Omron CX-Programmer project NewProject (CX-Programmer 9.75)

# PLC NewPLC1: CQM1H CPU51

## Global symbols (name address type ; comment)
1.00 BOOL  ; Manual/Automatic
1.08 BOOL  ; MAN/Forward
1.09 BOOL  ; MAN/Revrese
1.12 BOOL  ; Man/Rotate Right
1.13 BOOL  ; Man/Rotate Left
1.14 BOOL  ; Man/Piston Up
1.15 BOOL  ; Man/Piston Down
LR4.01 BOOL  ; MEM/Forward
LR4.02 BOOL  ; MEM/Reverse
LR4.05 BOOL  ; MEM/Rotate Right
LR4.06 BOOL  ; MEM/Rotate Left
LR4.07 BOOL  ; MEM/Piston Up
LR4.08 BOOL  ; MEM/Piston Down

## Program NewProgram1 (no task)

### Section Section1

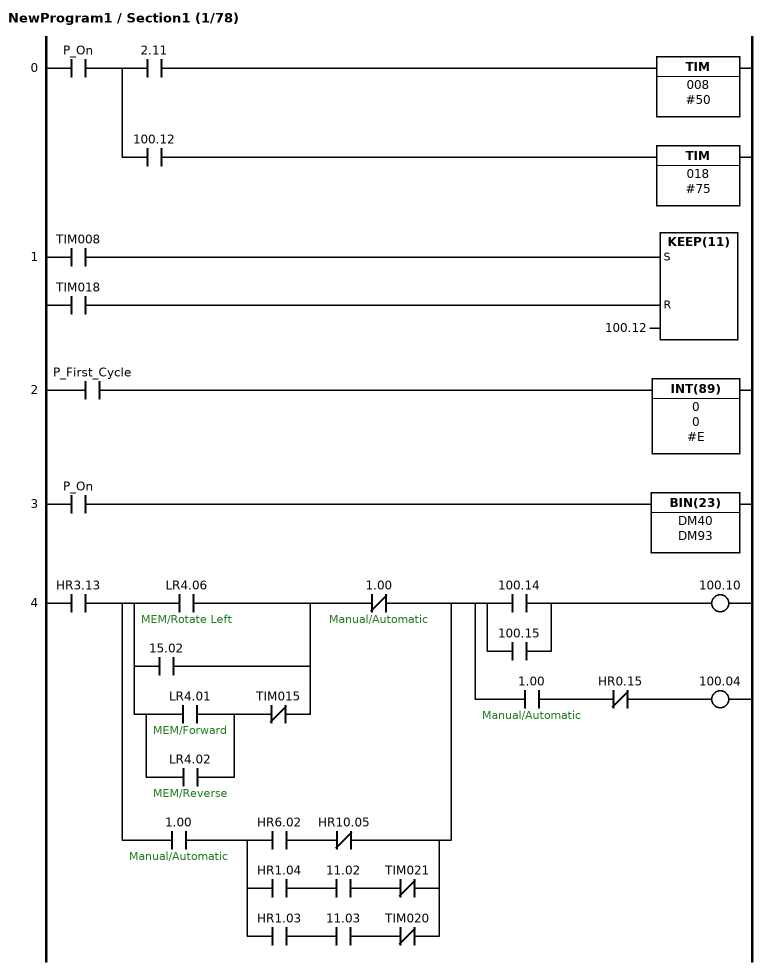
; rung 0
LD P_On
OUT TR0
AND 2.11
TIM 008 #50
LD TR0
AND 100.12
TIM 018 #75
; rung 1
LD TIM008
LD TIM018
KEEP(11) 100.12
; rung 2
LD P_First_Cycle
INT(89) 0 0 #E
; rung 3
LD P_On
BIN(23) DM40 DM93
; rung 4
LD HR3.13
LD LR4.06  ; MEM/Rotate Left
OR 15.02
LD LR4.01  ; MEM/Forward
OR LR4.02  ; MEM/Reverse
ANDNOT TIM015
ORLD
ANDNOT 1.00  ; Manual/Automatic
LD 1.00  ; Manual/Automatic
LD HR6.02
ANDNOT HR10.05
LD HR1.04
AND 11.02
ANDNOT TIM021
ORLD
LD HR1.03
AND 11.03
ANDNOT TIM020
ORLD
ANDLD
ORLD
ANDLD
OUT TR0
LD 100.14
OR 100.15
ANDLD
OUT 100.10
LD TR0
AND 1.00  ; Manual/Automatic
ANDNOT HR0.15
OUT 100.04

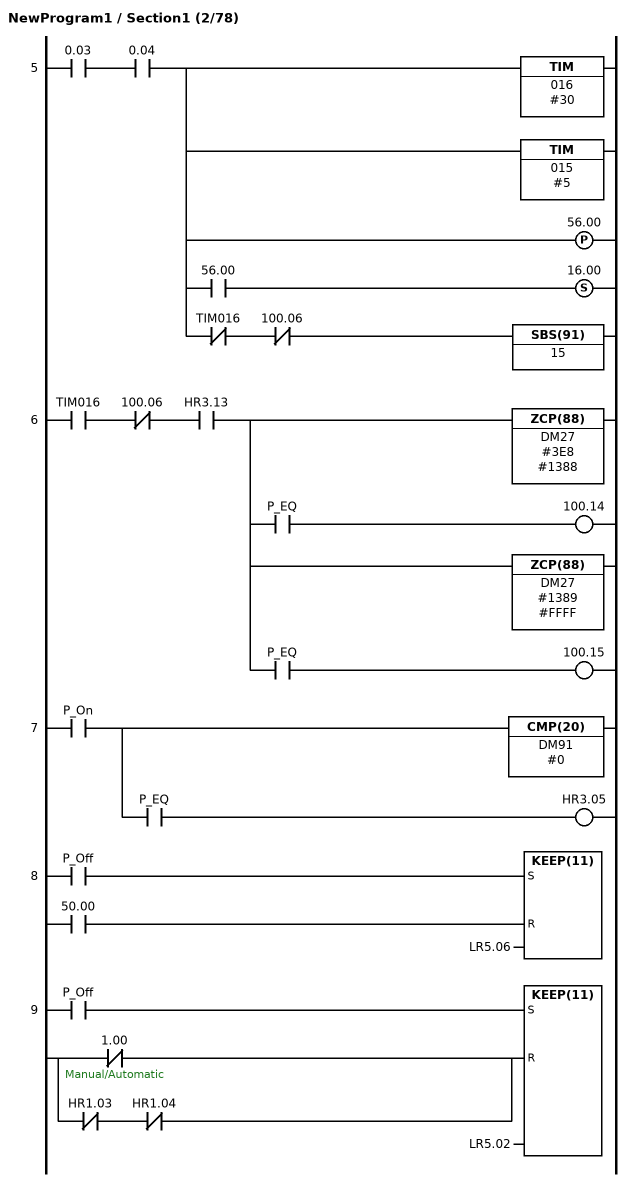
; rung 5
LD 0.03
AND 0.04
OUT TR0
TIM 016 #30
TIM 015 #5
DIFU(13) 56.00
AND 56.00
SET 16.00
LD TR0
ANDNOT TIM016
ANDNOT 100.06
SBS(91) 15
; rung 6
LD TIM016
ANDNOT 100.06
AND HR3.13
OUT TR0
ZCP(88) DM27 #3E8 #1388
AND P_EQ
OUT 100.14
LD TR0
ZCP(88) DM27 #1389 #FFFF
AND P_EQ
OUT 100.15
; rung 7
LD P_On
CMP(20) DM91 #0
AND P_EQ
OUT HR3.05
; rung 8
LD P_Off
LD 50.00
KEEP(11) LR5.06
; rung 9
LD P_Off
LDNOT 1.00  ; Manual/Automatic
LDNOT HR1.03
ANDNOT HR1.04
ORLD
KEEP(11) LR5.02

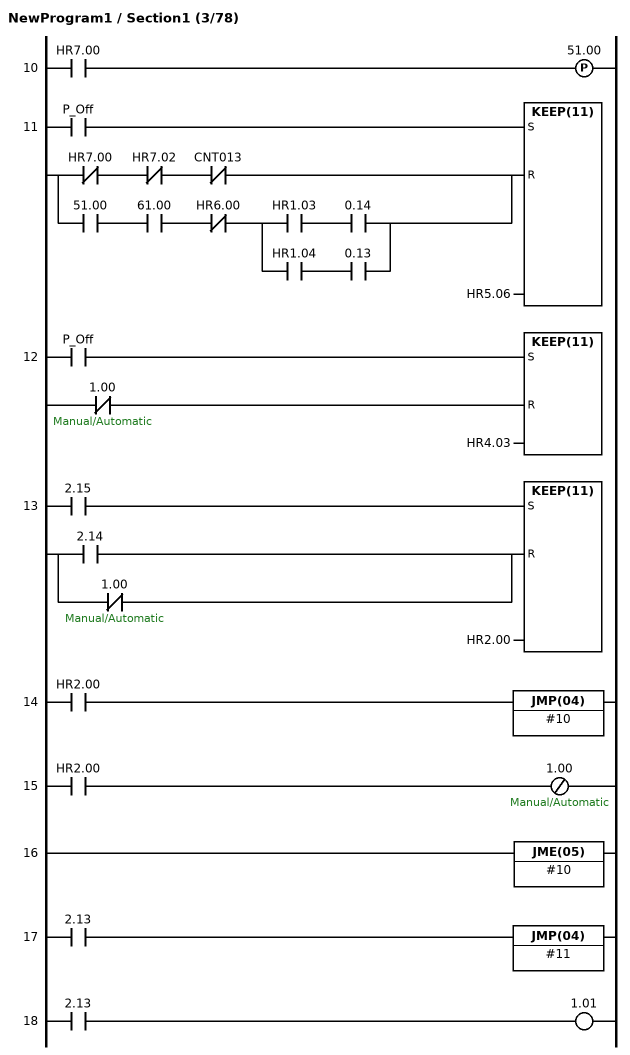
; rung 10
LD HR7.00
DIFU(13) 51.00
; rung 11
LD P_Off
LDNOT HR7.00
ANDNOT HR7.02
ANDNOT CNT013
LD 51.00
AND 61.00
ANDNOT HR6.00
LD HR1.03
AND 0.14
LD HR1.04
AND 0.13
ORLD
ANDLD
ORLD
KEEP(11) HR5.06
; rung 12
LD P_Off
LDNOT 1.00  ; Manual/Automatic
KEEP(11) HR4.03
; rung 13
LD 2.15
LD 2.14
ORNOT 1.00  ; Manual/Automatic
KEEP(11) HR2.00
; rung 14
LD HR2.00
JMP(04) #10
; rung 15
LD HR2.00
OUTNOT 1.00  ; Manual/Automatic
; rung 16
JME(05) #10
; rung 17
LD 2.13
JMP(04) #11
; rung 18
LD 2.13
OUT 1.01

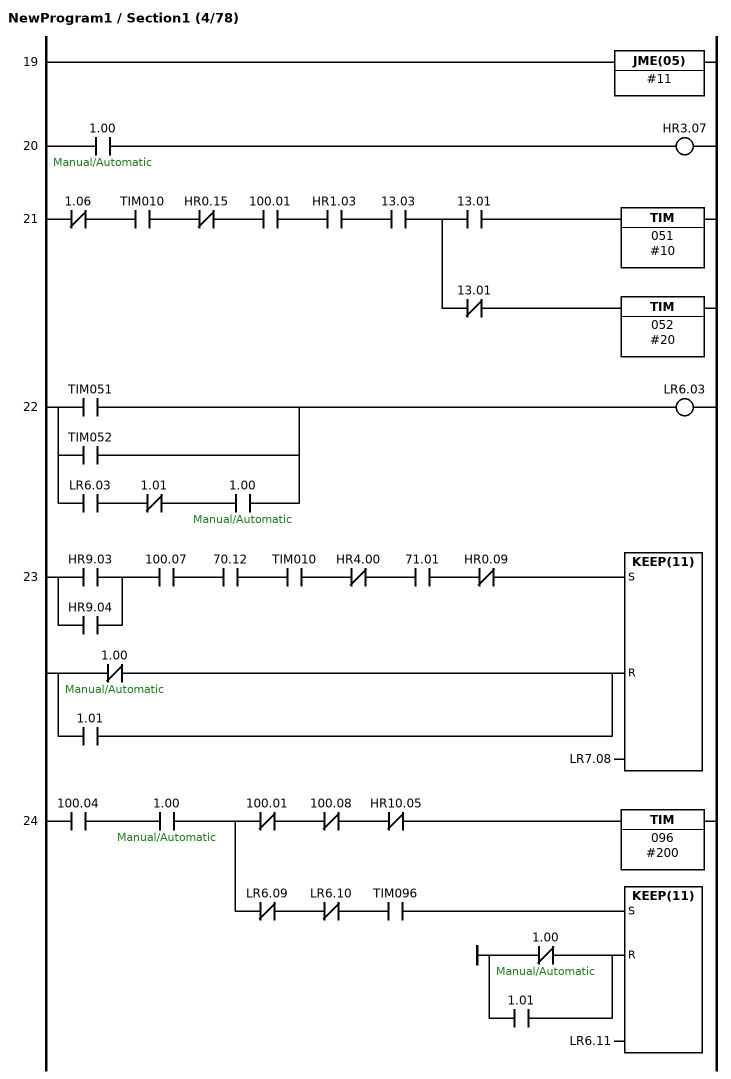
; rung 19
JME(05) #11
; rung 20
LD 1.00  ; Manual/Automatic
OUT HR3.07
; rung 21
LDNOT 1.06
AND TIM010
ANDNOT HR0.15
AND 100.01
AND HR1.03
AND 13.03
OUT TR0
AND 13.01
TIM 051 #10
LD TR0
ANDNOT 13.01
TIM 052 #20
; rung 22
LD TIM051
OR TIM052
LD LR6.03
ANDNOT 1.01
AND 1.00  ; Manual/Automatic
ORLD
OUT LR6.03
; rung 23
LD HR9.03
OR HR9.04
AND 100.07
AND 70.12
AND TIM010
ANDNOT HR4.00
AND 71.01
ANDNOT HR0.09
LDNOT 1.00  ; Manual/Automatic
OR 1.01
KEEP(11) LR7.08
; rung 24
LD 100.04
AND 1.00  ; Manual/Automatic
OUT TR0
ANDNOT 100.01
ANDNOT 100.08
ANDNOT HR10.05
TIM 096 #200
LD TR0
ANDNOT LR6.09
ANDNOT LR6.10
AND TIM096
LDNOT 1.00  ; Manual/Automatic
OR 1.01
KEEP(11) LR6.11

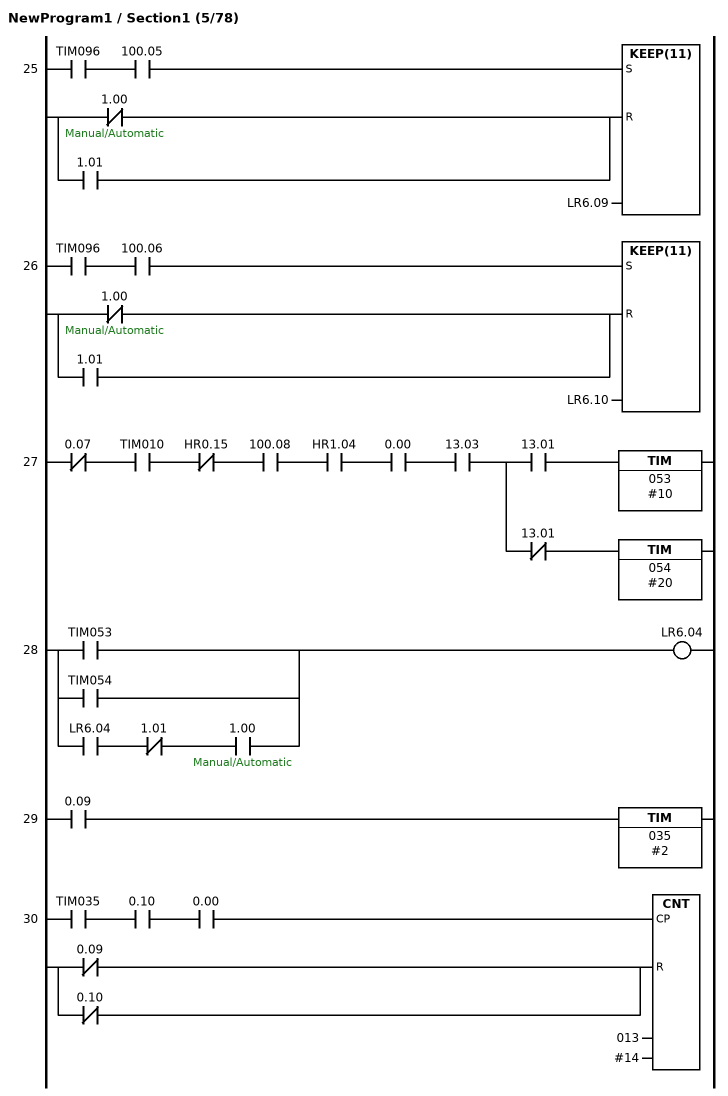
; rung 25
LD TIM096
AND 100.05
LDNOT 1.00  ; Manual/Automatic
OR 1.01
KEEP(11) LR6.09
; rung 26
LD TIM096
AND 100.06
LDNOT 1.00  ; Manual/Automatic
OR 1.01
KEEP(11) LR6.10
; rung 27
LDNOT 0.07
AND TIM010
ANDNOT HR0.15
AND 100.08
AND HR1.04
AND 0.00
AND 13.03
OUT TR0
AND 13.01
TIM 053 #10
LD TR0
ANDNOT 13.01
TIM 054 #20
; rung 28
LD TIM053
OR TIM054
LD LR6.04
ANDNOT 1.01
AND 1.00  ; Manual/Automatic
ORLD
OUT LR6.04
; rung 29
LD 0.09
TIM 035 #2
; rung 30
LD TIM035
AND 0.10
AND 0.00
LDNOT 0.09
ORNOT 0.10
CNT 013 #14

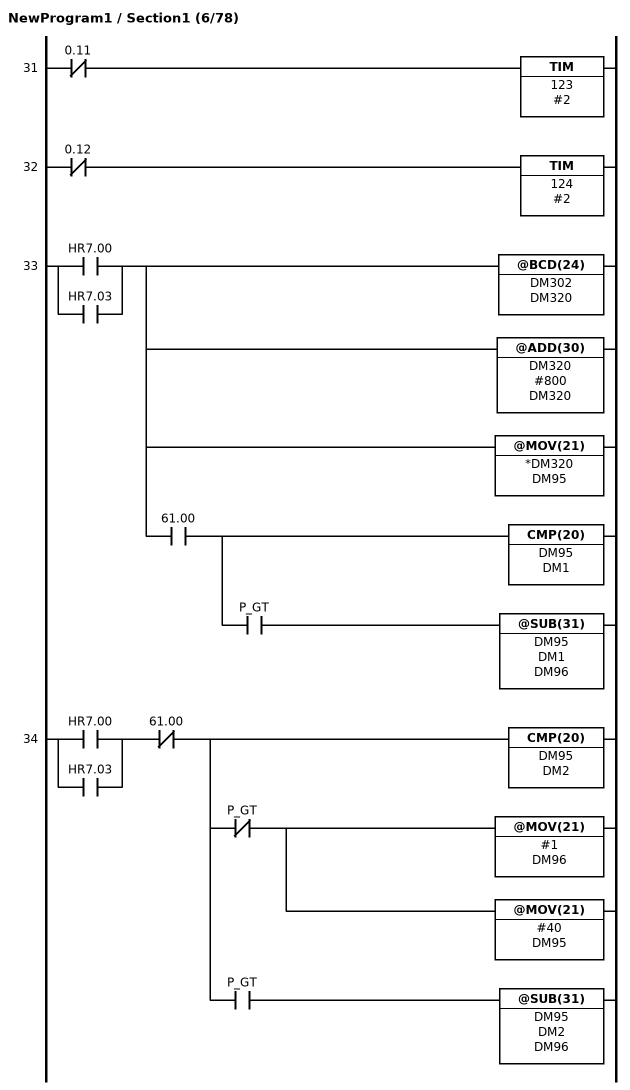
; rung 31
LDNOT 0.11
TIM 123 #2
; rung 32
LDNOT 0.12
TIM 124 #2
; rung 33
LD HR7.00
OR HR7.03
@BCD(24) DM302 DM320
@ADD(30) DM320 #800 DM320
@MOV(21) *DM320 DM95
AND 61.00
CMP(20) DM95 DM1
AND P_GT
@SUB(31) DM95 DM1 DM96
; rung 34
LD HR7.00
OR HR7.03
ANDNOT 61.00
OUT TR0
CMP(20) DM95 DM2
ANDNOT P_GT
@MOV(21) #1 DM96
@MOV(21) #40 DM95
LD TR0
AND P_GT
@SUB(31) DM95 DM2 DM96

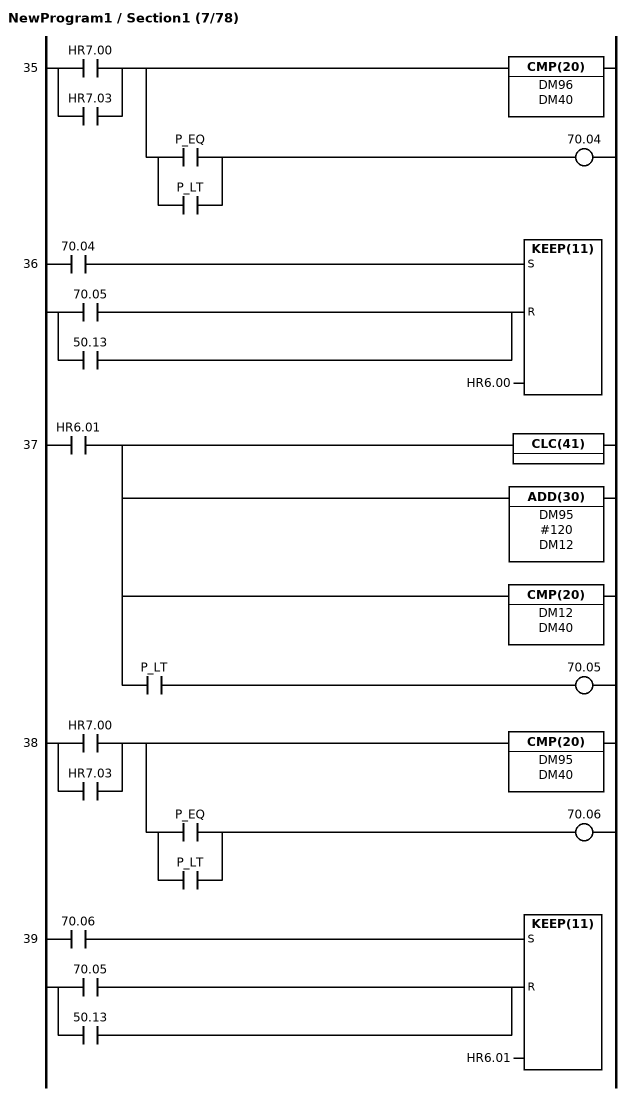
; rung 35
LD HR7.00
OR HR7.03
CMP(20) DM96 DM40
LD P_EQ
OR P_LT
ANDLD
OUT 70.04
; rung 36
LD 70.04
LD 70.05
OR 50.13
KEEP(11) HR6.00
; rung 37
LD HR6.01
CLC(41)
ADD(30) DM95 #120 DM12
CMP(20) DM12 DM40
AND P_LT
OUT 70.05
; rung 38
LD HR7.00
OR HR7.03
CMP(20) DM95 DM40
LD P_EQ
OR P_LT
ANDLD
OUT 70.06
; rung 39
LD 70.06
LD 70.05
OR 50.13
KEEP(11) HR6.01

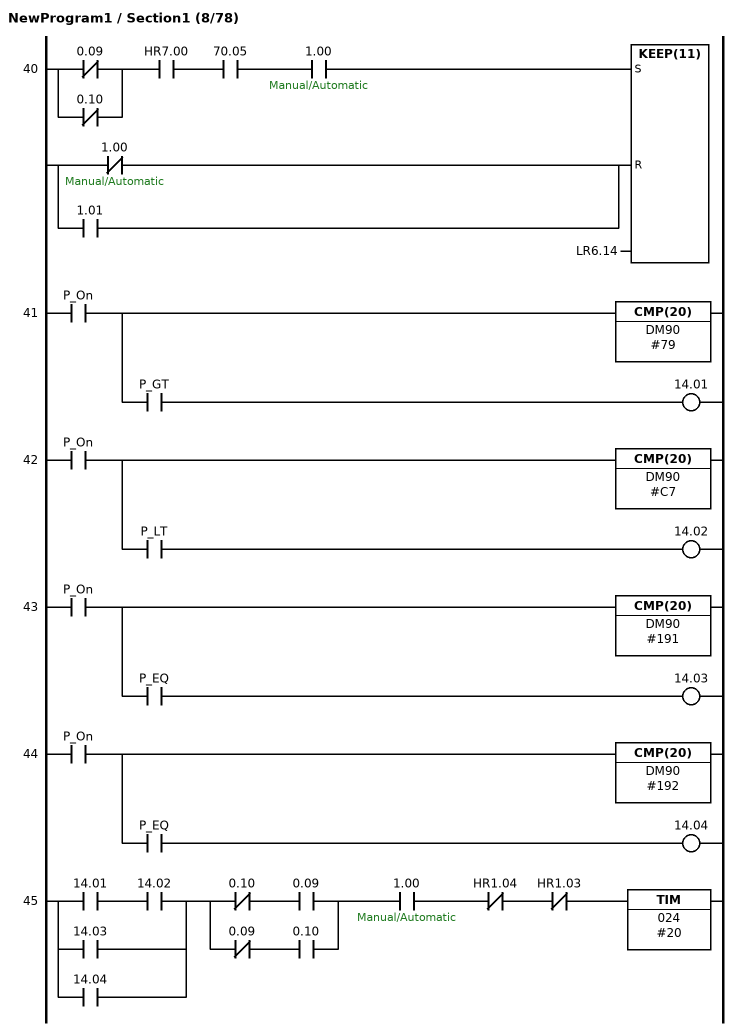
; rung 40
LDNOT 0.09
ORNOT 0.10
AND HR7.00
AND 70.05
AND 1.00  ; Manual/Automatic
LDNOT 1.00  ; Manual/Automatic
OR 1.01
KEEP(11) LR6.14
; rung 41
LD P_On
CMP(20) DM90 #79
AND P_GT
OUT 14.01
; rung 42
LD P_On
CMP(20) DM90 #C7
AND P_LT
OUT 14.02
; rung 43
LD P_On
CMP(20) DM90 #191
AND P_EQ
OUT 14.03
; rung 44
LD P_On
CMP(20) DM90 #192
AND P_EQ
OUT 14.04
; rung 45
LD 14.01
AND 14.02
OR 14.03
OR 14.04
LDNOT 0.10
AND 0.09
LDNOT 0.09
AND 0.10
ORLD
ANDLD
AND 1.00  ; Manual/Automatic
ANDNOT HR1.04
ANDNOT HR1.03
TIM 024 #20

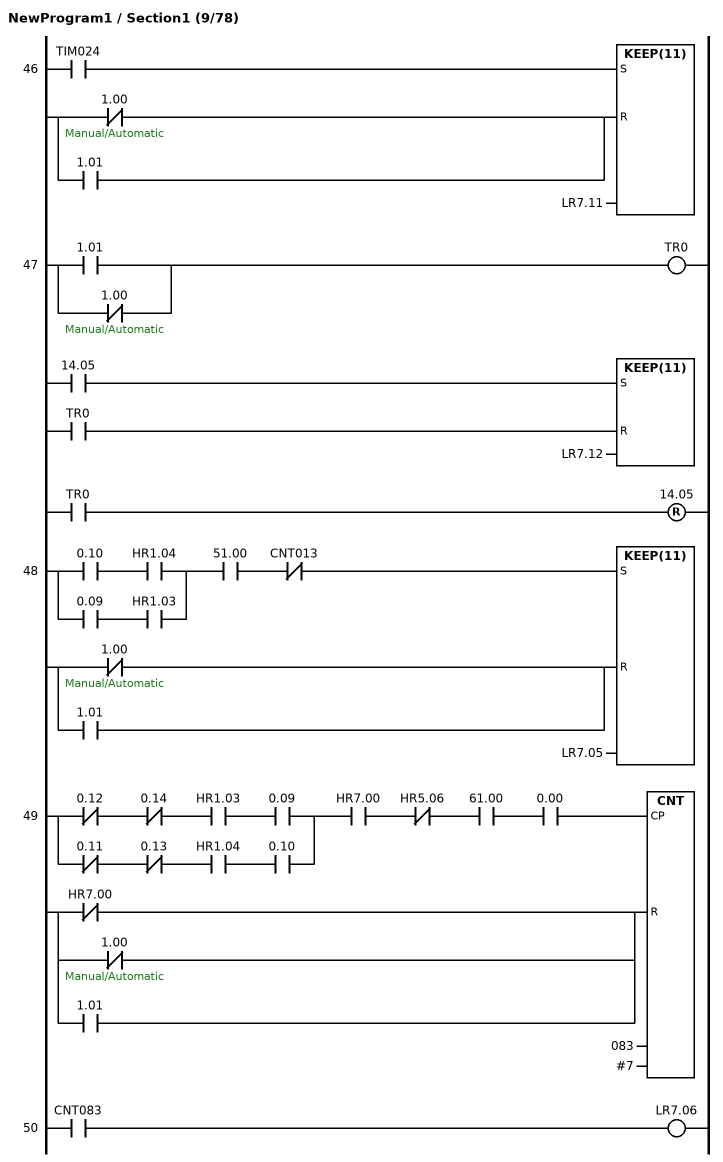
; rung 46
LD TIM024
LDNOT 1.00  ; Manual/Automatic
OR 1.01
KEEP(11) LR7.11
; rung 47
LD 14.05
LD 1.01
ORNOT 1.00  ; Manual/Automatic
OUT TR0
KEEP(11) LR7.12
LD TR0
RSET 14.05
; rung 48
LD 0.10
AND HR1.04
LD 0.09
AND HR1.03
ORLD
AND 51.00
ANDNOT CNT013
LDNOT 1.00  ; Manual/Automatic
OR 1.01
KEEP(11) LR7.05
; rung 49
LDNOT 0.12
ANDNOT 0.14
AND HR1.03
AND 0.09
LDNOT 0.11
ANDNOT 0.13
AND HR1.04
AND 0.10
ORLD
AND HR7.00
ANDNOT HR5.06
AND 61.00
AND 0.00
LDNOT HR7.00
ORNOT 1.00  ; Manual/Automatic
OR 1.01
CNT 083 #7
; rung 50
LD CNT083
OUT LR7.06

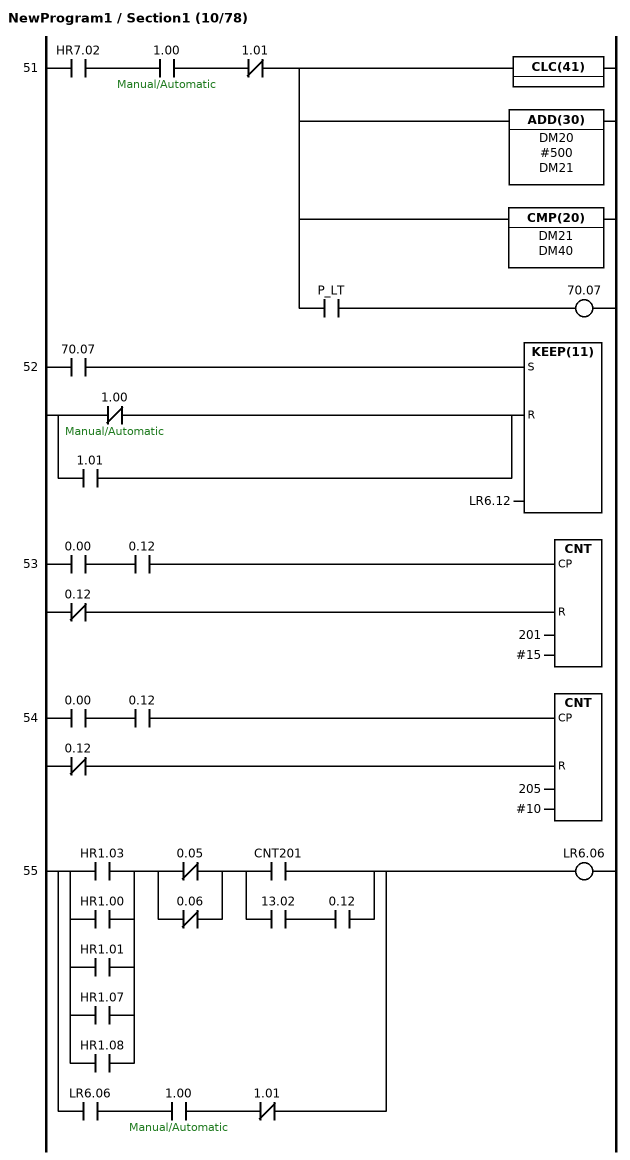
; rung 51
LD HR7.02
AND 1.00  ; Manual/Automatic
ANDNOT 1.01
CLC(41)
ADD(30) DM20 #500 DM21
CMP(20) DM21 DM40
AND P_LT
OUT 70.07
; rung 52
LD 70.07
LDNOT 1.00  ; Manual/Automatic
OR 1.01
KEEP(11) LR6.12
; rung 53
LD 0.00
AND 0.12
LDNOT 0.12
CNT 201 #15
; rung 54
LD 0.00
AND 0.12
LDNOT 0.12
CNT 205 #10
; rung 55
LD HR1.03
OR HR1.00
OR HR1.01
OR HR1.07
OR HR1.08
LDNOT 0.05
ORNOT 0.06
ANDLD
LD CNT201
LD 13.02
AND 0.12
ORLD
ANDLD
LD LR6.06
AND 1.00  ; Manual/Automatic
ANDNOT 1.01
ORLD
OUT LR6.06

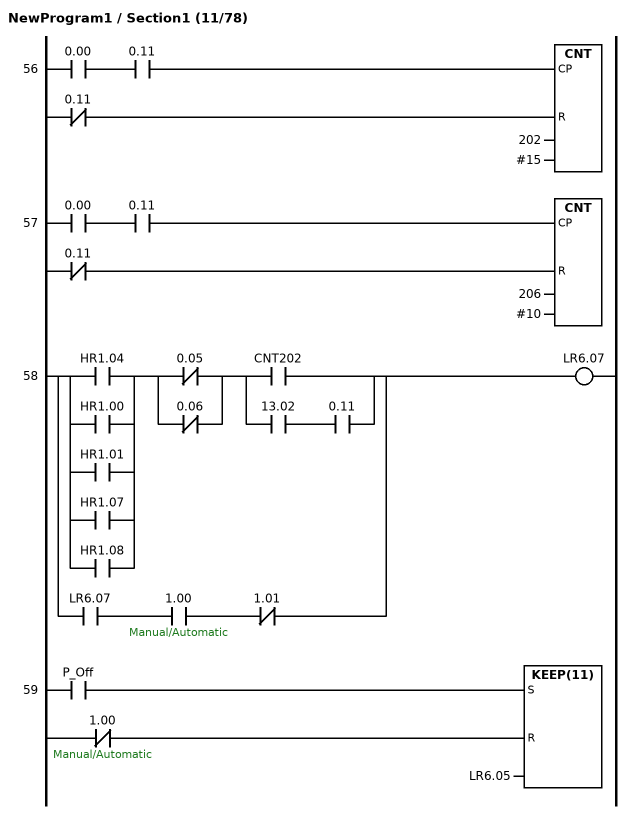
; rung 56
LD 0.00
AND 0.11
LDNOT 0.11
CNT 202 #15
; rung 57
LD 0.00
AND 0.11
LDNOT 0.11
CNT 206 #10
; rung 58
LD HR1.04
OR HR1.00
OR HR1.01
OR HR1.07
OR HR1.08
LDNOT 0.05
ORNOT 0.06
ANDLD
LD CNT202
LD 13.02
AND 0.11
ORLD
ANDLD
LD LR6.07
AND 1.00  ; Manual/Automatic
ANDNOT 1.01
ORLD
OUT LR6.07
; rung 59
LD P_Off
LDNOT 1.00  ; Manual/Automatic
KEEP(11) LR6.05

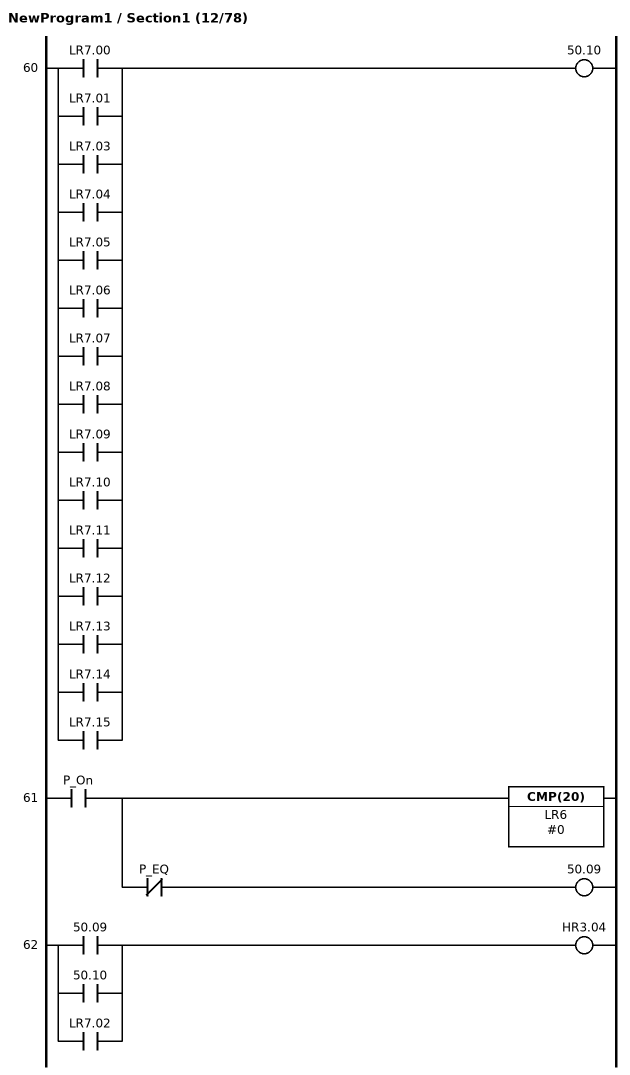
; rung 60
LD LR7.00
OR LR7.01
OR LR7.03
OR LR7.04
OR LR7.05
OR LR7.06
OR LR7.07
OR LR7.08
OR LR7.09
OR LR7.10
OR LR7.11
OR LR7.12
OR LR7.13
OR LR7.14
OR LR7.15
OUT 50.10
; rung 61
LD P_On
CMP(20) LR6 #0
ANDNOT P_EQ
OUT 50.09
; rung 62
LD 50.09
OR 50.10
OR LR7.02
OUT HR3.04

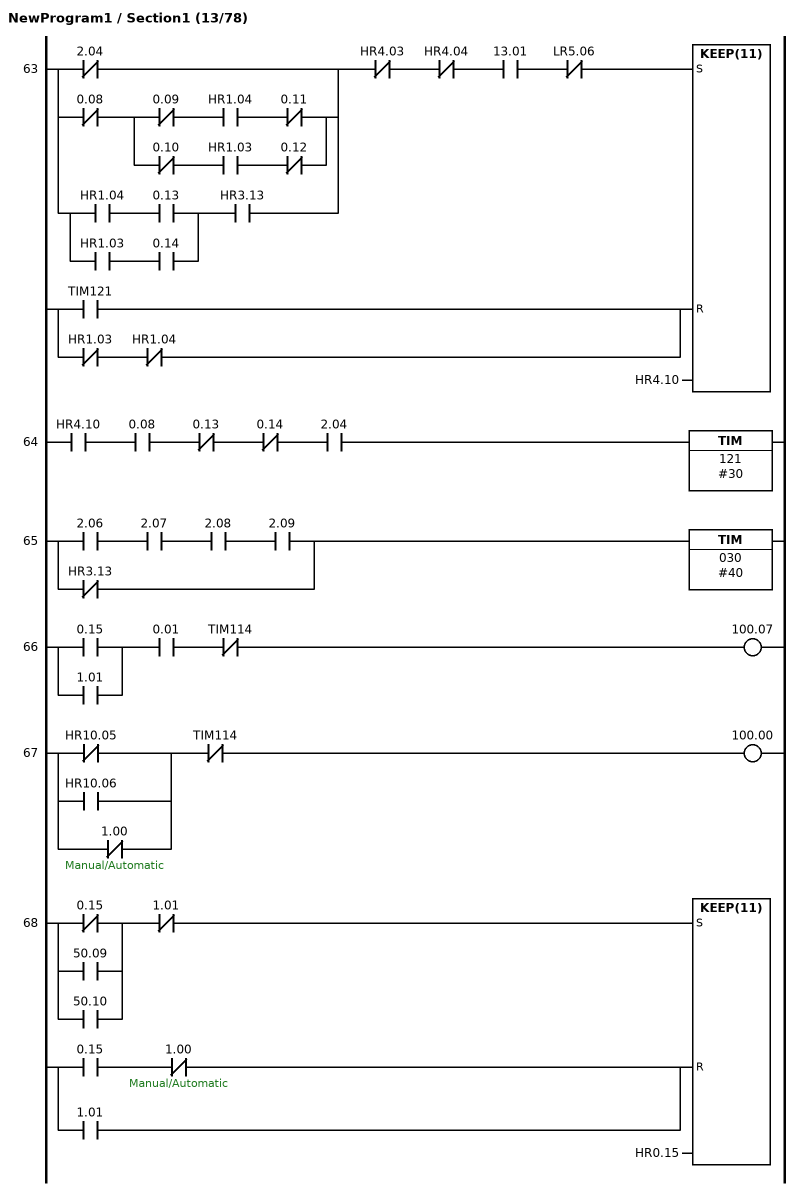
; rung 63
LDNOT 2.04
LDNOT 0.08
LDNOT 0.09
AND HR1.04
ANDNOT 0.11
LDNOT 0.10
AND HR1.03
ANDNOT 0.12
ORLD
ANDLD
ORLD
LD HR1.04
AND 0.13
LD HR1.03
AND 0.14
ORLD
AND HR3.13
ORLD
ANDNOT HR4.03
ANDNOT HR4.04
AND 13.01
ANDNOT LR5.06
LD TIM121
LDNOT HR1.03
ANDNOT HR1.04
ORLD
KEEP(11) HR4.10
; rung 64
LD HR4.10
AND 0.08
ANDNOT 0.13
ANDNOT 0.14
AND 2.04
TIM 121 #30
; rung 65
LD 2.06
AND 2.07
AND 2.08
AND 2.09
ORNOT HR3.13
TIM 030 #40
; rung 66
LD 0.15
OR 1.01
AND 0.01
ANDNOT TIM114
OUT 100.07
; rung 67
LDNOT HR10.05
OR HR10.06
ORNOT 1.00  ; Manual/Automatic
ANDNOT TIM114
OUT 100.00
; rung 68
LDNOT 0.15
OR 50.09
OR 50.10
ANDNOT 1.01
LD 0.15
ANDNOT 1.00  ; Manual/Automatic
OR 1.01
KEEP(11) HR0.15

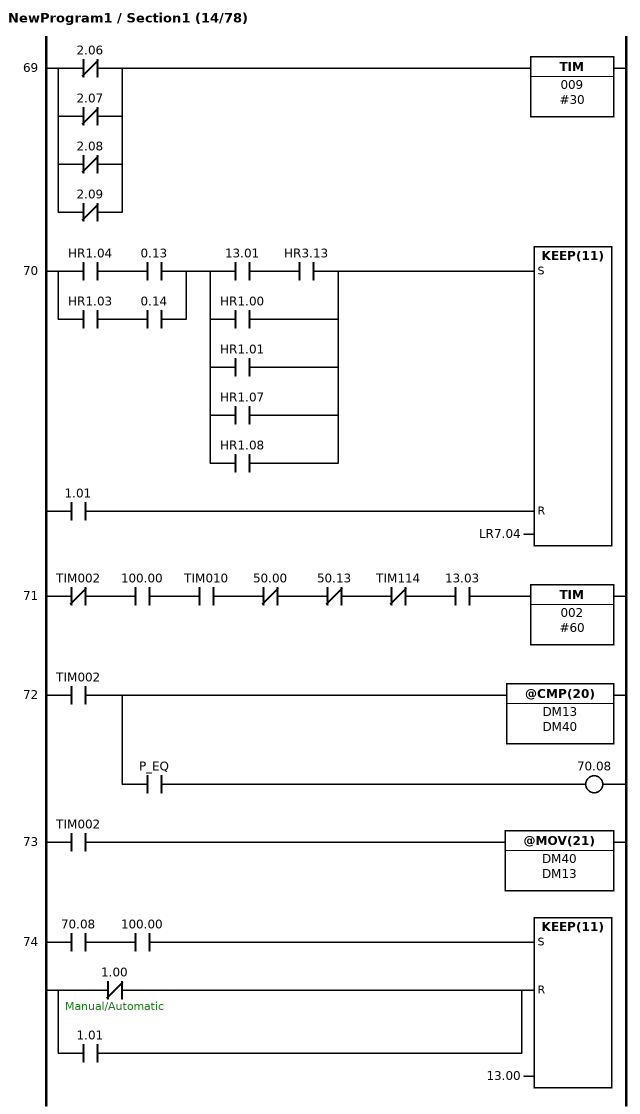
; rung 69
LDNOT 2.06
ORNOT 2.07
ORNOT 2.08
ORNOT 2.09
TIM 009 #30
; rung 70
LD HR1.04
AND 0.13
LD HR1.03
AND 0.14
ORLD
LD 13.01
AND HR3.13
OR HR1.00
OR HR1.01
OR HR1.07
OR HR1.08
ANDLD
LD 1.01
KEEP(11) LR7.04
; rung 71
LDNOT TIM002
AND 100.00
AND TIM010
ANDNOT 50.00
ANDNOT 50.13
ANDNOT TIM114
AND 13.03
TIM 002 #60
; rung 72
LD TIM002
@CMP(20) DM13 DM40
AND P_EQ
OUT 70.08
; rung 73
LD TIM002
@MOV(21) DM40 DM13
; rung 74
LD 70.08
AND 100.00
LDNOT 1.00  ; Manual/Automatic
OR 1.01
KEEP(11) 13.00

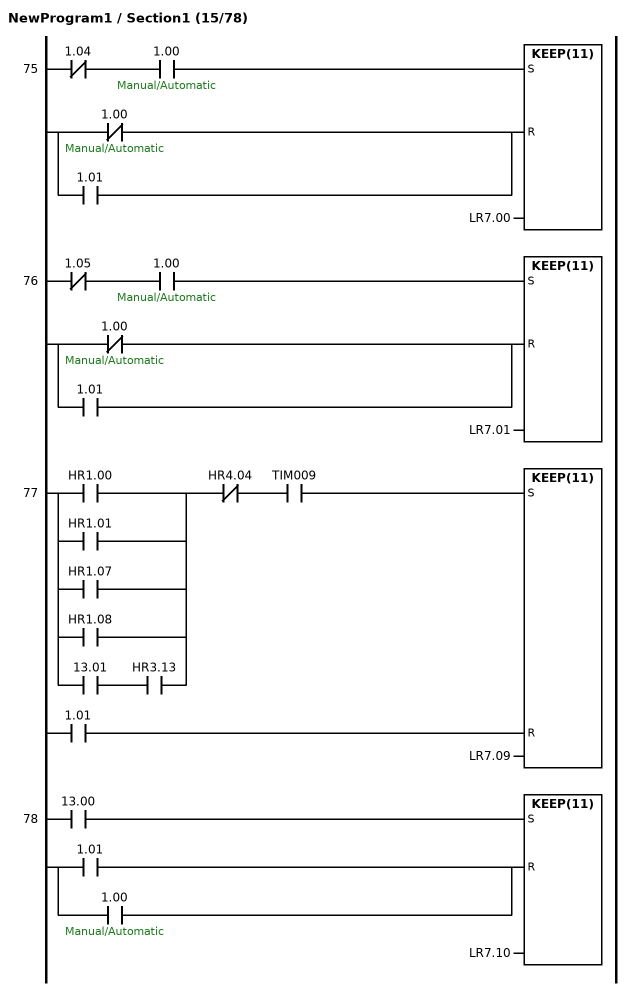
; rung 75
LDNOT 1.04
AND 1.00  ; Manual/Automatic
LDNOT 1.00  ; Manual/Automatic
OR 1.01
KEEP(11) LR7.00
; rung 76
LDNOT 1.05
AND 1.00  ; Manual/Automatic
LDNOT 1.00  ; Manual/Automatic
OR 1.01
KEEP(11) LR7.01
; rung 77
LD HR1.00
OR HR1.01
OR HR1.07
OR HR1.08
LD 13.01
AND HR3.13
ORLD
ANDNOT HR4.04
AND TIM009
LD 1.01
KEEP(11) LR7.09
; rung 78
LD 13.00
LD 1.01
OR 1.00  ; Manual/Automatic
KEEP(11) LR7.10

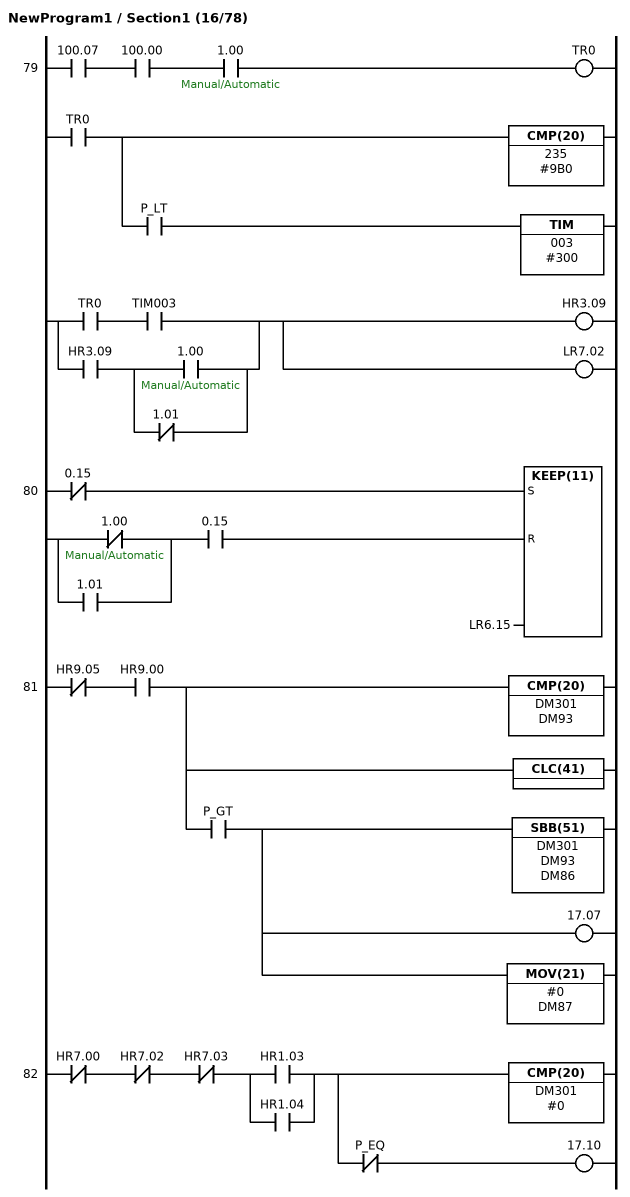
; rung 79
LD 100.07
AND 100.00
AND 1.00  ; Manual/Automatic
OUT TR0
CMP(20) 235 #9B0
AND P_LT
TIM 003 #300
LD TR0
AND TIM003
LD HR3.09
LD 1.00  ; Manual/Automatic
ORNOT 1.01
ANDLD
ORLD
OUT HR3.09
OUT LR7.02
; rung 80
LDNOT 0.15
LDNOT 1.00  ; Manual/Automatic
OR 1.01
AND 0.15
KEEP(11) LR6.15
; rung 81
LDNOT HR9.05
AND HR9.00
CMP(20) DM301 DM93
CLC(41)
AND P_GT
SBB(51) DM301 DM93 DM86
OUT 17.07
MOV(21) #0 DM87
; rung 82
LDNOT HR7.00
ANDNOT HR7.02
ANDNOT HR7.03
LD HR1.03
OR HR1.04
ANDLD
CMP(20) DM301 #0
ANDNOT P_EQ
OUT 17.10

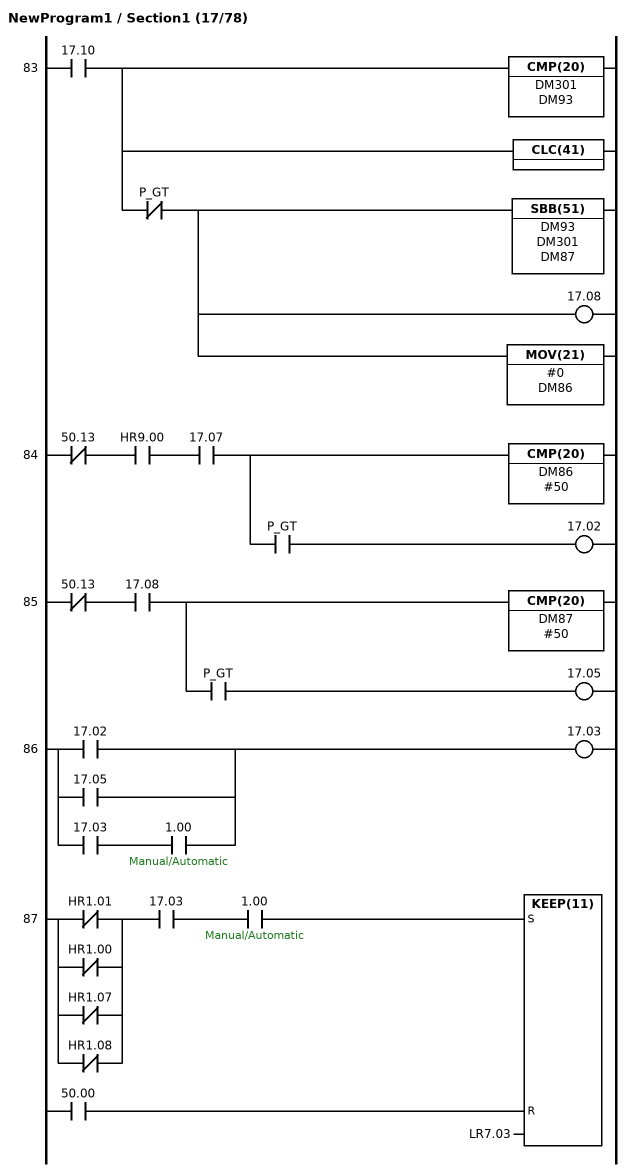
; rung 83
LD 17.10
CMP(20) DM301 DM93
CLC(41)
ANDNOT P_GT
SBB(51) DM93 DM301 DM87
OUT 17.08
MOV(21) #0 DM86
; rung 84
LDNOT 50.13
AND HR9.00
AND 17.07
CMP(20) DM86 #50
AND P_GT
OUT 17.02
; rung 85
LDNOT 50.13
AND 17.08
CMP(20) DM87 #50
AND P_GT
OUT 17.05
; rung 86
LD 17.02
OR 17.05
LD 17.03
AND 1.00  ; Manual/Automatic
ORLD
OUT 17.03
; rung 87
LDNOT HR1.01
ORNOT HR1.00
ORNOT HR1.07
ORNOT HR1.08
AND 17.03
AND 1.00  ; Manual/Automatic
LD 50.00
KEEP(11) LR7.03

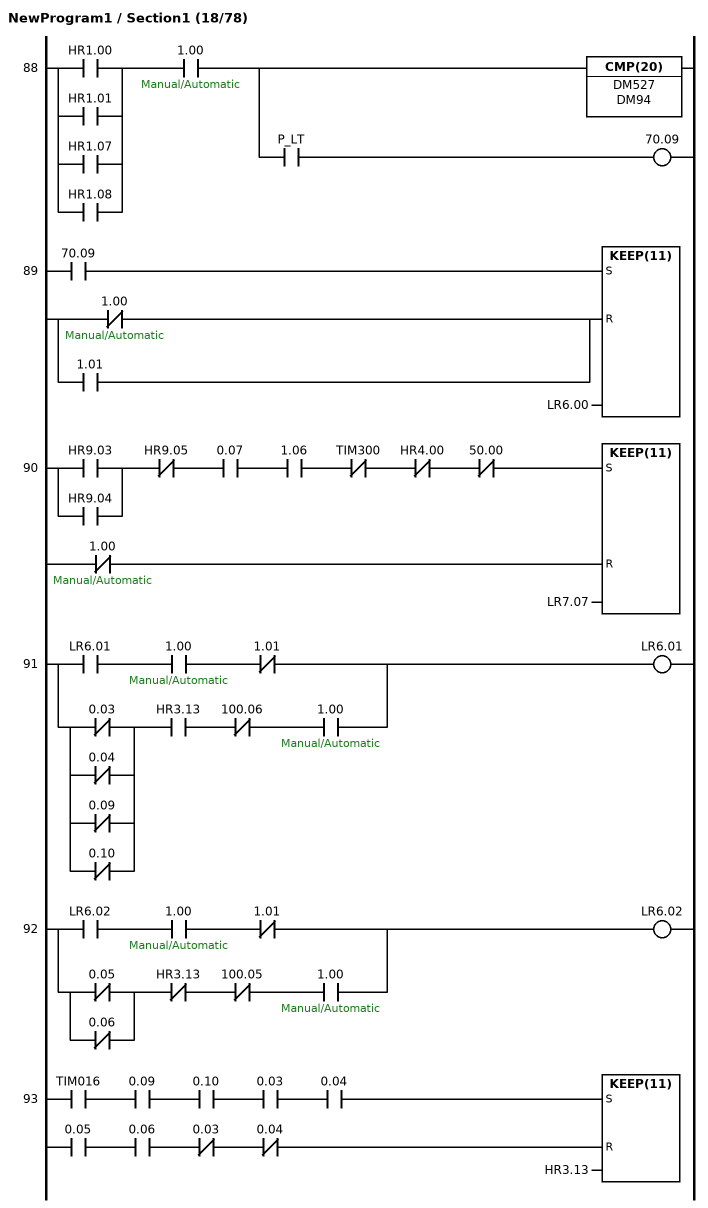
; rung 88
LD HR1.00
OR HR1.01
OR HR1.07
OR HR1.08
AND 1.00  ; Manual/Automatic
CMP(20) DM527 DM94
AND P_LT
OUT 70.09
; rung 89
LD 70.09
LDNOT 1.00  ; Manual/Automatic
OR 1.01
KEEP(11) LR6.00
; rung 90
LD HR9.03
OR HR9.04
ANDNOT HR9.05
AND 0.07
AND 1.06
ANDNOT TIM300
ANDNOT HR4.00
ANDNOT 50.00
LDNOT 1.00  ; Manual/Automatic
KEEP(11) LR7.07
; rung 91
LD LR6.01
AND 1.00  ; Manual/Automatic
ANDNOT 1.01
LDNOT 0.03
ORNOT 0.04
ORNOT 0.09
ORNOT 0.10
AND HR3.13
ANDNOT 100.06
AND 1.00  ; Manual/Automatic
ORLD
OUT LR6.01
; rung 92
LD LR6.02
AND 1.00  ; Manual/Automatic
ANDNOT 1.01
LDNOT 0.05
ORNOT 0.06
ANDNOT HR3.13
ANDNOT 100.05
AND 1.00  ; Manual/Automatic
ORLD
OUT LR6.02
; rung 93
LD TIM016
AND 0.09
AND 0.10
AND 0.03
AND 0.04
LD 0.05
AND 0.06
ANDNOT 0.03
ANDNOT 0.04
KEEP(11) HR3.13

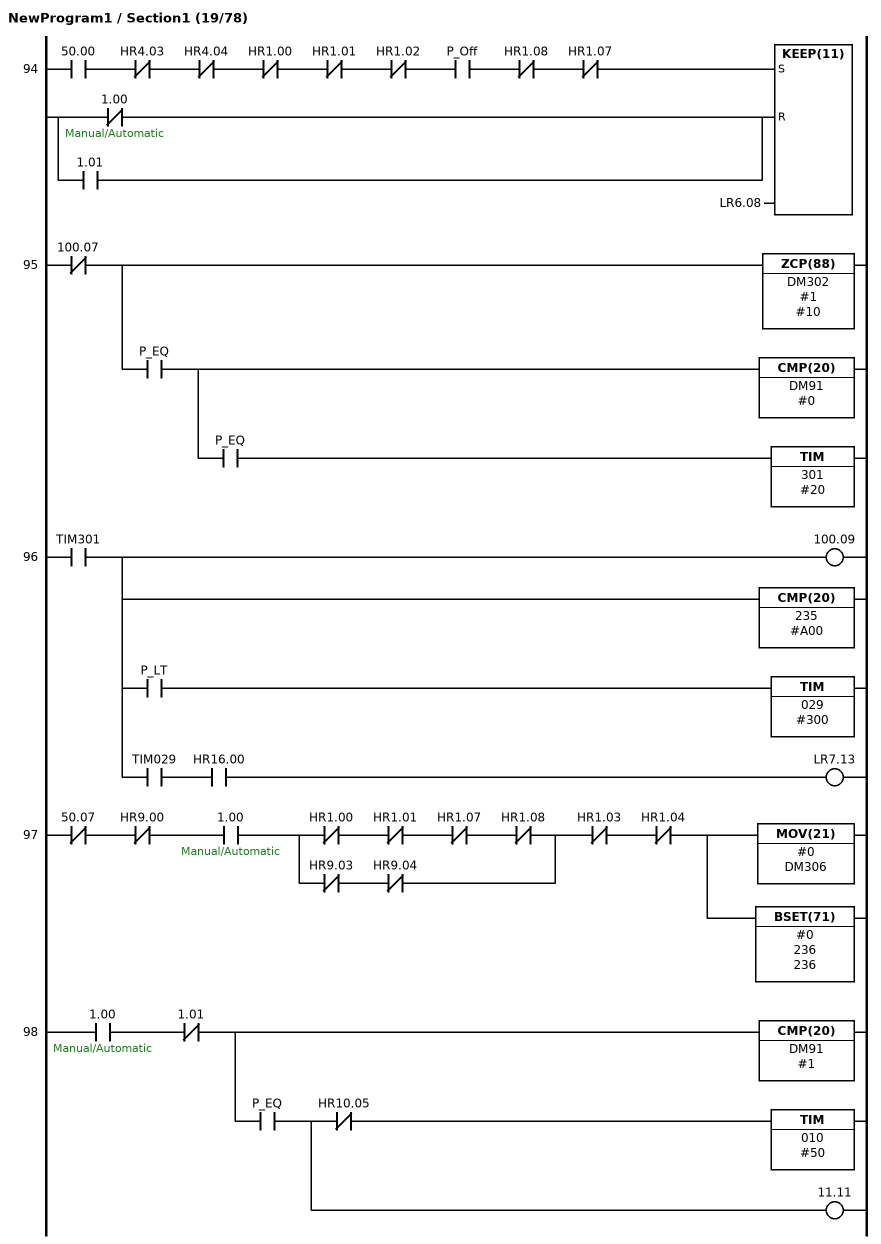
; rung 94
LD 50.00
ANDNOT HR4.03
ANDNOT HR4.04
ANDNOT HR1.00
ANDNOT HR1.01
ANDNOT HR1.02
AND P_Off
ANDNOT HR1.08
ANDNOT HR1.07
LDNOT 1.00  ; Manual/Automatic
OR 1.01
KEEP(11) LR6.08
; rung 95
LDNOT 100.07
ZCP(88) DM302 #1 #10
AND P_EQ
CMP(20) DM91 #0
AND P_EQ
TIM 301 #20
; rung 96
LD TIM301
OUT TR0
OUT 100.09
CMP(20) 235 #A00
AND P_LT
TIM 029 #300
LD TR0
AND TIM029
AND HR16.00
OUT LR7.13
; rung 97
LDNOT 50.07
ANDNOT HR9.00
AND 1.00  ; Manual/Automatic
LDNOT HR1.00
ANDNOT HR1.01
ANDNOT HR1.07
ANDNOT HR1.08
LDNOT HR9.03
ANDNOT HR9.04
ORLD
ANDLD
ANDNOT HR1.03
ANDNOT HR1.04
MOV(21) #0 DM306
BSET(71) #0 236 236
; rung 98
LD 1.00  ; Manual/Automatic
ANDNOT 1.01
CMP(20) DM91 #1
AND P_EQ
OUT TR0
ANDNOT HR10.05
TIM 010 #50
LD TR0
OUT 11.11

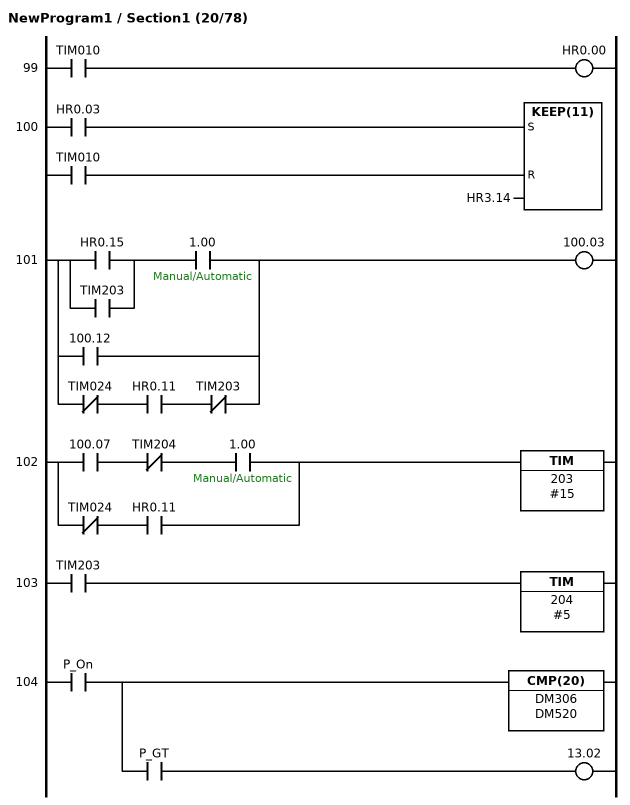
; rung 99
LD TIM010
OUT HR0.00
; rung 100
LD HR0.03
LD TIM010
KEEP(11) HR3.14
; rung 101
LD HR0.15
OR TIM203
AND 1.00  ; Manual/Automatic
OR 100.12
LDNOT TIM024
AND HR0.11
ANDNOT TIM203
ORLD
OUT 100.03
; rung 102
LD 100.07
ANDNOT TIM204
AND 1.00  ; Manual/Automatic
LDNOT TIM024
AND HR0.11
ORLD
TIM 203 #15
; rung 103
LD TIM203
TIM 204 #5
; rung 104
LD P_On
CMP(20) DM306 DM520
AND P_GT
OUT 13.02

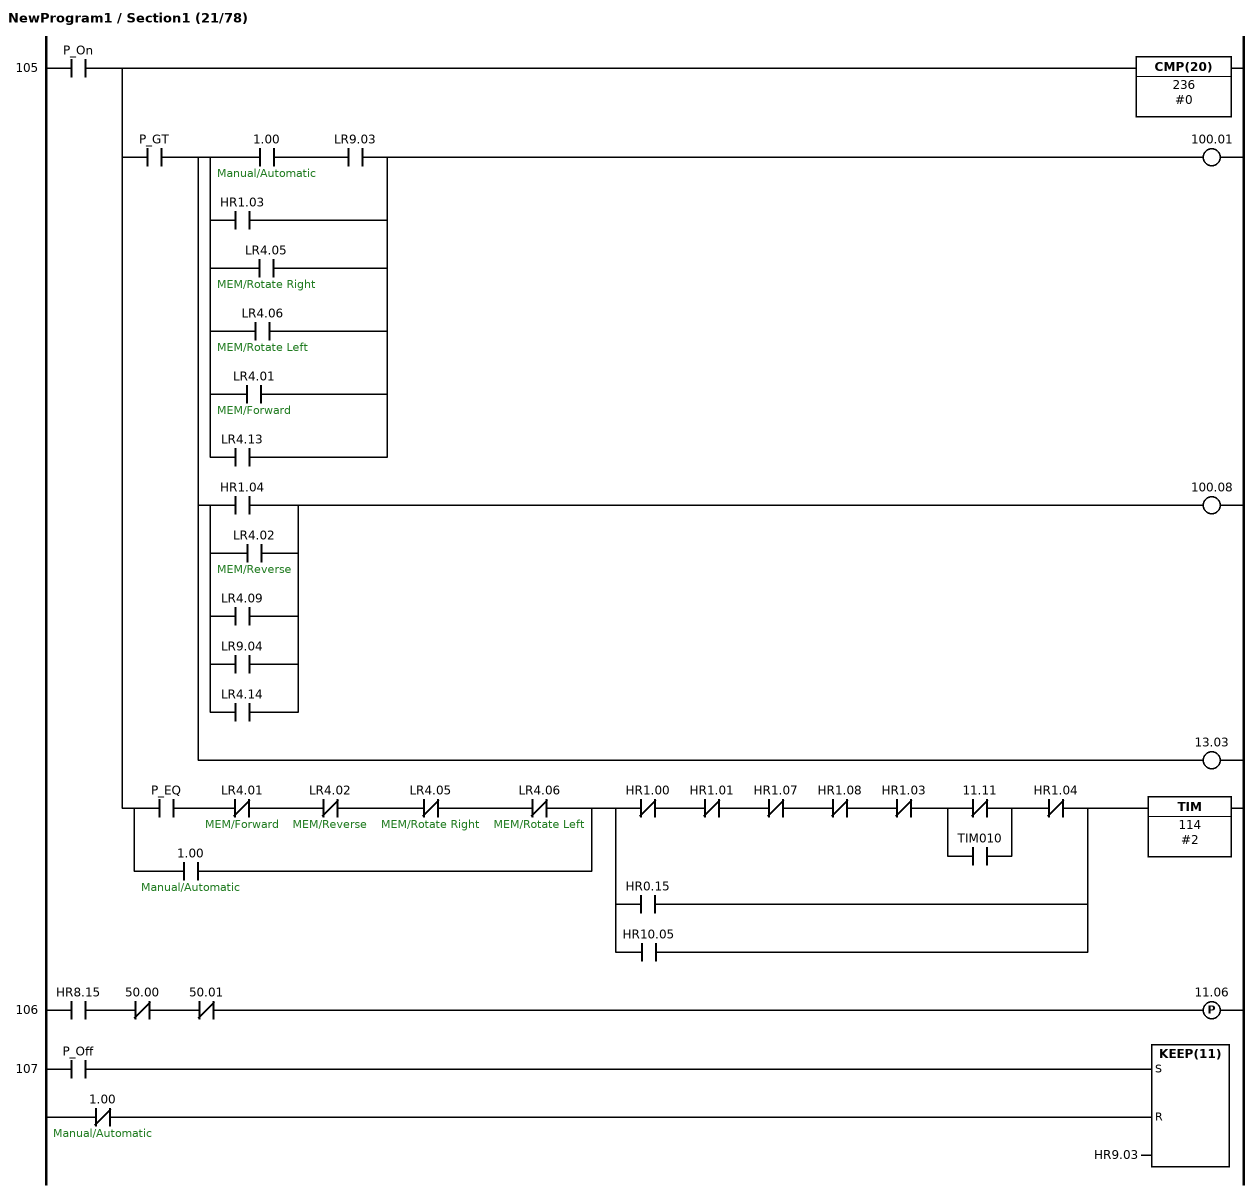
; rung 105
LD P_On
OUT TR0
CMP(20) 236 #0
AND P_GT
OUT TR1
LD 1.00  ; Manual/Automatic
AND LR9.03
OR HR1.03
OR LR4.05  ; MEM/Rotate Right
OR LR4.06  ; MEM/Rotate Left
OR LR4.01  ; MEM/Forward
OR LR4.13
ANDLD
OUT 100.01
LD TR1
LD HR1.04
OR LR4.02  ; MEM/Reverse
OR LR4.09
OR LR9.04
OR LR4.14
ANDLD
OUT 100.08
LD TR1
OUT 13.03
LD TR0
LD P_EQ
ANDNOT LR4.01  ; MEM/Forward
ANDNOT LR4.02  ; MEM/Reverse
ANDNOT LR4.05  ; MEM/Rotate Right
ANDNOT LR4.06  ; MEM/Rotate Left
OR 1.00  ; Manual/Automatic
ANDLD
LDNOT HR1.00
ANDNOT HR1.01
ANDNOT HR1.07
ANDNOT HR1.08
ANDNOT HR1.03
LDNOT 11.11
OR TIM010
ANDLD
ANDNOT HR1.04
OR HR0.15
OR HR10.05
ANDLD
TIM 114 #2
; rung 106
LD HR8.15
ANDNOT 50.00
ANDNOT 50.01
DIFU(13) 11.06
; rung 107
LD P_Off
LDNOT 1.00  ; Manual/Automatic
KEEP(11) HR9.03

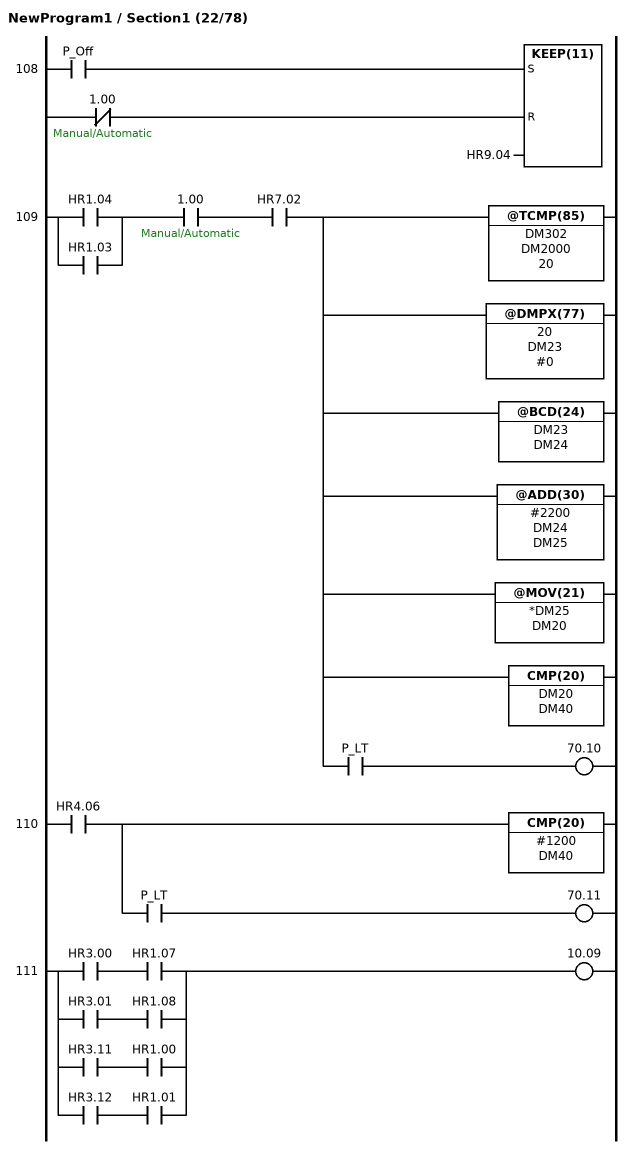
; rung 108
LD P_Off
LDNOT 1.00  ; Manual/Automatic
KEEP(11) HR9.04
; rung 109
LD HR1.04
OR HR1.03
AND 1.00  ; Manual/Automatic
AND HR7.02
@TCMP(85) DM302 DM2000 20
@DMPX(77) 20 DM23 #0
@BCD(24) DM23 DM24
@ADD(30) #2200 DM24 DM25
@MOV(21) *DM25 DM20
CMP(20) DM20 DM40
AND P_LT
OUT 70.10
; rung 110
LD HR4.06
CMP(20) #1200 DM40
AND P_LT
OUT 70.11
; rung 111
LD HR3.00
AND HR1.07
LD HR3.01
AND HR1.08
ORLD
LD HR3.11
AND HR1.00
ORLD
LD HR3.12
AND HR1.01
ORLD
OUT 10.09

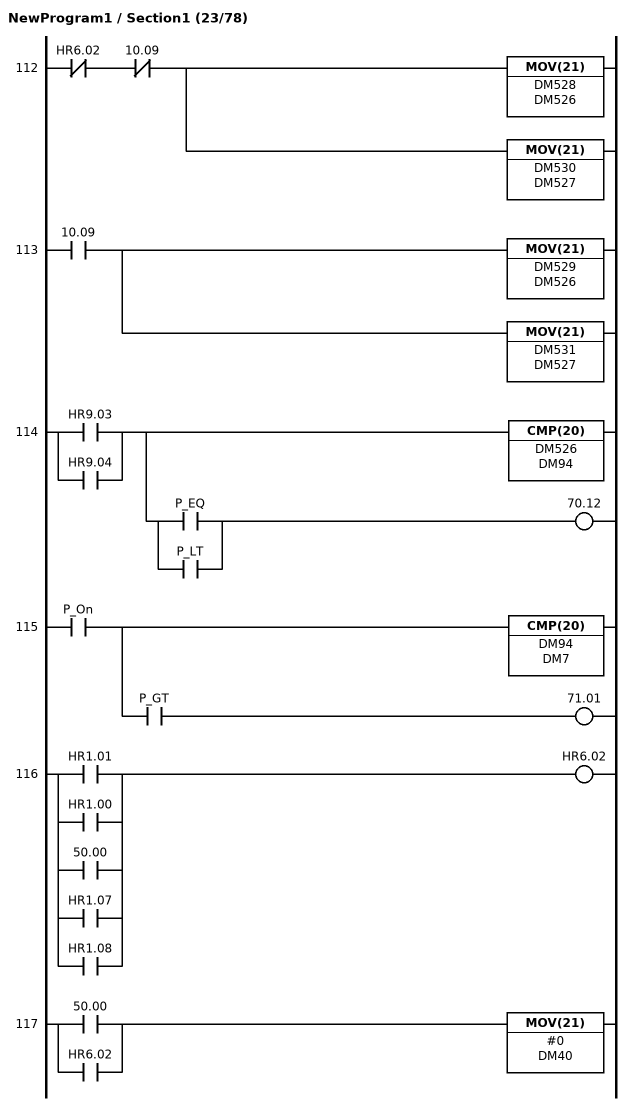
; rung 112
LDNOT HR6.02
ANDNOT 10.09
MOV(21) DM528 DM526
MOV(21) DM530 DM527
; rung 113
LD 10.09
MOV(21) DM529 DM526
MOV(21) DM531 DM527
; rung 114
LD HR9.03
OR HR9.04
CMP(20) DM526 DM94
LD P_EQ
OR P_LT
ANDLD
OUT 70.12
; rung 115
LD P_On
CMP(20) DM94 DM7
AND P_GT
OUT 71.01
; rung 116
LD HR1.01
OR HR1.00
OR 50.00
OR HR1.07
OR HR1.08
OUT HR6.02
; rung 117
LD 50.00
OR HR6.02
MOV(21) #0 DM40

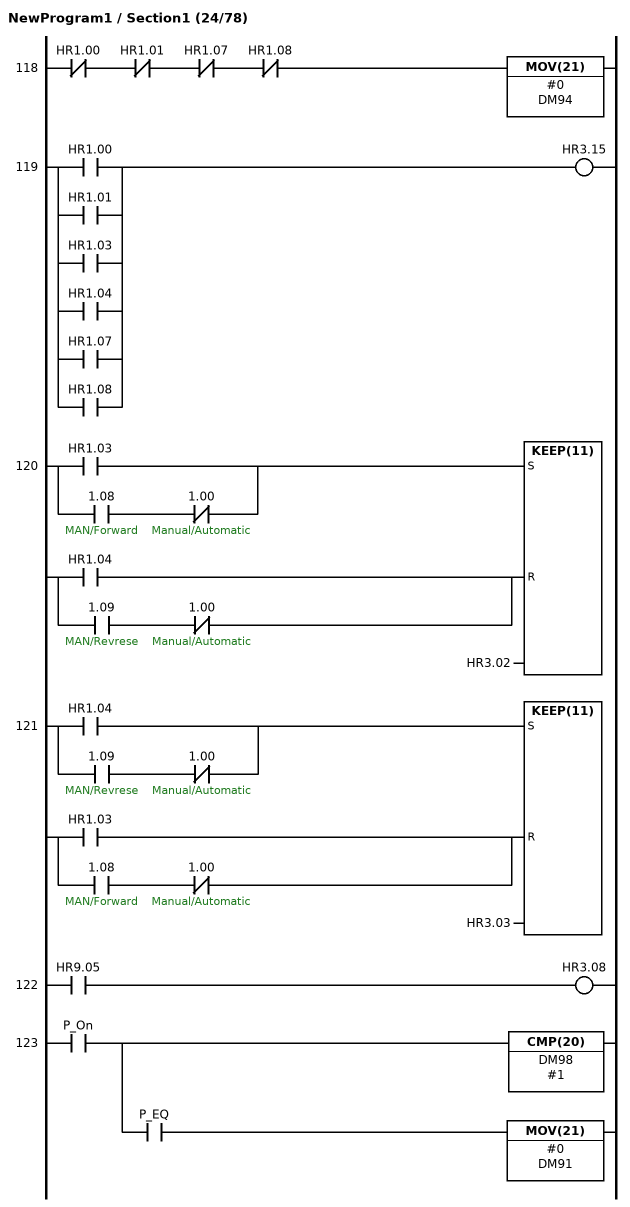
; rung 118
LDNOT HR1.00
ANDNOT HR1.01
ANDNOT HR1.07
ANDNOT HR1.08
MOV(21) #0 DM94
; rung 119
LD HR1.00
OR HR1.01
OR HR1.03
OR HR1.04
OR HR1.07
OR HR1.08
OUT HR3.15
; rung 120
LD HR1.03
LD 1.08  ; MAN/Forward
ANDNOT 1.00  ; Manual/Automatic
ORLD
LD HR1.04
LD 1.09  ; MAN/Revrese
ANDNOT 1.00  ; Manual/Automatic
ORLD
KEEP(11) HR3.02
; rung 121
LD HR1.04
LD 1.09  ; MAN/Revrese
ANDNOT 1.00  ; Manual/Automatic
ORLD
LD HR1.03
LD 1.08  ; MAN/Forward
ANDNOT 1.00  ; Manual/Automatic
ORLD
KEEP(11) HR3.03
; rung 122
LD HR9.05
OUT HR3.08
; rung 123
LD P_On
CMP(20) DM98 #1
AND P_EQ
MOV(21) #0 DM91

